// TwinCAT 3 PLC project Plc1_AmeClient
// ProgramVersion: 3.1.4024.0
// libraries:
//   Tc2_Standard, * (Beckhoff Automation GmbH)
//   Tc2_System, * (Beckhoff Automation GmbH)
//   Tc2_TcpIp, * (Beckhoff Automation GmbH)
//   Tc3_Module, * (Beckhoff Automation GmbH)
// project tree:
//   / PlcTask.TcTTO
//   POUs/AmeClient/ AmeClient.TcPOU (not stored), AmeClientParam.TcGVL (not stored)
//   POUs/AmeClient/DUTs/AssyMethods/ St_Assy_Base.TcDUT (not stored), St_Assy_Complete.TcDUT (not stored), St_Assy_GetDetails.TcDUT (not stored), St_Assy_SetParametricsAndNCNative.TcDUT (not stored), St_Assy_SetReferences.TcDUT (not stored), St_Assy_SignOff.TcDUT (not stored), St_Assy_Start.TcDUT (not stored)
//   POUs/AmeClient/DUTs/ E_AssyComplete.TcDUT (not stored)
//   POUs/ MAIN.TcPOU
//   POUs/OOP/ I_Command.TcIO (not stored), I_Device.TcIO (not stored), Stereo.TcPOU, TurnOffCommand.TcPOU (not stored), TurnOnCommand.TcPOU (not stored)
// real-time tasks:
//   TASK PlcTask: cycle T#10ms, priority 20, ADS port 350
// motion (NC):
//   TASK NC-Task 1 SAF: cycle T#2ms, priority 4, ADS port 501
//   TASK NC-Task 1 SVB: cycle T#10ms, priority 8, ADS port 511
//   AXIS Axis 1 (id 1)
//     OtherSettings: AllowMotionCmdToSlave=true
//     encoder EncType=19
//       EncPara: MaxCount=#xffffffff
//     drive DrvType=16
//       DrvPara: MaxCount=#xffffffff
//         Analog: TorqueSetpointScale=10, ScaleFactorActTorque=0.1
//         TimeComp: TaskDelayCycles=1
//     controller CtrType=1
//       CtrPara: PriorControlFactor=1
//         Observer: BandWidth=20
// I/O:
//   DEVICE Device 1 (EtherCAT) (disabled), AmsNetId 192.168.48.2.2.1
//     Term 1 (EK1100) [EK1100 EtherCAT Coupler (2A E-Bus)]
//       Term 2 (EL6631) [EL6631 PROFINET IO Controller]
//     ServoControllerX (CMMT-AS-MP-S1) [CMMT-AS-MP-S1]
//   DEVICE Device 2 (EL6631) (disabled), AmsNetId 192.168.48.2.3.1
//     tcpniodevice [Beckhoff Automation TwinCAT PLC PROFINET I/O Device with I/Os, V2.43, PROFIenergy supported; 1 port TwinCAT PN Device]
//       modules: Term 1 (DAP Module)
//     tcpniodevice-4 [Beckhoff Automation TwinCAT PLC PROFINET I/O Device with I/Os, V2.32, 1 port diagnostic supported TwinCAT PN Device]
//       modules: Term 2 (DAP Module), Term 3 (8 Word Output), Term 4 (2 Word Output), Term 5 (1 Word Output), Term 6 (1 Word Output), Term 7 (8 Word Input), Term 8 (2 Word Input), Term 9 (8 Word Input), Term 10 (64 Word Input)
// variable links:
//   (this object) <-> Device 1 (EtherCAT)/ServoControllerX (CMMT-AS-MP-S1)
//     Drive/Inputs/In/nDataIn3[0] <-> Inputs/Torque actual value
//     Drive/Inputs/In/nDcOutputTime <-> InfoData/DcOutputShift
//     Drive/Inputs/In/nState1 <-> Inputs/Statusword
//     Drive/Inputs/In/nState2 <-> Inputs/Statusword @bit 8
//     Drive/Inputs/In/nState4 @bit 1 <-> WcState/InputToggle
//     Drive/Inputs/In/nState4 <-> WcState/WcState
//     Drive/Inputs/In/nState5 <-> Inputs/Modes of operation display
//     Drive/Outputs/Out/nCtrl1 <-> Outputs/Controlword
//     Drive/Outputs/Out/nCtrl2 <-> Outputs/Controlword @bit 8
//     Drive/Outputs/Out/nCtrl5 <-> Outputs/Modes of operation
//     Drive/Outputs/Out/nDataOut1 <-> Outputs/Target position
//     Drive/Outputs/Out/nDataOut2 <-> Outputs/Target velocity
//     Drive/Outputs/Out/nDataOut3[0] <-> Outputs/Torque offset
//     Drive/Outputs/Out/nDataOut4[0] <-> Outputs/Target torque
//     Enc/Inputs/In/nDataIn1 <-> Inputs/Position actual value
//     Enc/Inputs/In/nDataIn7 <-> Inputs/Velocity actual value
//     Enc/Inputs/In/nDcInputTime <-> InfoData/DcInputShift
//     Enc/Inputs/In/nState4 @bit 1 <-> WcState/InputToggle
//     Enc/Inputs/In/nState4 <-> WcState/WcState

CONFIGURATION Plc1_AmeClient
    RESOURCE PLC ON TwinCAT3
        TASK PlcTask(INTERVAL := T#10ms, PRIORITY := 20);
        PROGRAM MAIN WITH PlcTask : MAIN;
    END_RESOURCE
END_CONFIGURATION

// ---- POUs/MAIN.TcPOU
PROGRAM MAIN

VAR	

	AmeClient 							:AmeClient(iType := 1, sSrvNetId := '', sRemoteHost := '192.168.48.2', udiRemotePort := 2001, tTimeout := T#5S);
	_bAssy_GetDetails 					:BOOL;
	_st_Assy_GetDetails					: St_Assy_GetDetails := (sSfc := 'TEST0100000000001010184E0010', iOpIndex := 0); 
	_bAssy_Start						:BOOL;
	_st_Assy_Start						:St_Assy_Start := (sSfc := 'TEST0100000000001010184E0010', iOpIndex := 0);
	_bAssy_SetReferences				:BOOL;
	_st_Assy_SetReferences				:St_Assy_SetReferences := (sSfc := 'TEST0100000000001010184E0010', sCustomField :='PLASMA_COUNTER|0',  iOpIndex := 0);
	_bAssy_SetParametricsAndNCNative	:BOOL;
	_st_Assy_SetParametricsAndNCNative	:St_Assy_SetParametricsAndNCNative := (	sSfc 			:= 'TEST0100000000001010184E0010',
																				sProgramId 		:= 'PROGRAMID_TEST1',
																				sProgramRevision:= 'PROGRAMREVISION_TEST1',
																				sTestStep		:= 'TESTESTEP1', 
																				sDescription	:= 'DESCRIPTION1', 
																				sValue			:= 'TESTVALUE1', 
																				sUnit			:= 'UNIT1', 
																				sLowerLimit		:= 'LOWERLIMIT1', 
																				sUpperLimit		:= 'UPPERLIMIT1', 
																				sState			:= '0', 
																				sAdapter		:= '2',
																				iOpIndex 		:= 0);
	_bAssy_Complete						:BOOL;
	_st_Assy_Complete					:St_Assy_Complete := (sSfc := 'TEST0100000000001010184E0010', eState := E_AssyComplete.PASS, iOpIndex := 0);
	_bAssy_SignOff						:BOOL;
	_st_Assy_SignOff					:St_Assy_SignOff := (sSfc := 'TEST0100000000001010184E0010', iOpIndex := 0);
	_sSendMsg							:STRING(AmeClientParam.udiMSG_SIZE);
	_sRcvMsg							:STRING(AmeClientParam.udiMSG_SIZE);
	
END_VAR

VAR
	bMsg	:Bool;
END_VAR

// Assy GetDetails******************************************************

IF(_bAssy_GetDetails = TRUE AND_THEN AmeClient.Assy_GetDetails_1026(_st_Assy_GetDetails) = TRUE) THEN
	_bAssy_GetDetails := FALSE;
	_sSendMsg 		:= AmeClient.sSendMsg;
	_sRcvMsg 		:= AmeClient.sRcvMsg;
END_IF
//**********************************************************************

// Assy Start***********************************************************
IF(_bAssy_Start = TRUE AND_THEN AmeClient.Assy_Start(_st_Assy_Start) = TRUE) THEN
	_bAssy_Start := FALSE;
	_sSendMsg 	:= AmeClient.sSendMsg;
	_sRcvMsg 	:= AmeClient.sRcvMsg;
END_IF
//**********************************************************************

// Assy setReferences***************************************************
IF(_bAssy_SetReferences = TRUE AND_THEN AmeClient.Assy_SetReferences_3026(_st_Assy_SetReferences) = TRUE ) THEN
	_bAssy_SetReferences := FALSE;
	_sSendMsg 	:= AmeClient.sSendMsg;
	_sRcvMsg 	:= AmeClient.sRcvMsg;
END_IF
//**********************************************************************

// Assy SetParametricsAndNCNative***************************************
IF(_bAssy_SetParametricsAndNCNative = TRUE AND_THEN AmeClient.Assy_SetParametricsAndNCNative_3503(_st_Assy_SetParametricsAndNCNative) = TRUE) THEN
	_bAssy_SetParametricsAndNCNative := FALSE;
	_sSendMsg 	:= AmeClient.sSendMsg;
	_sRcvMsg 	:= AmeClient.sRcvMsg;
END_IF
//**********************************************************************

// Assy compleate*******************************************************
IF(_bAssy_Complete = TRUE AND_THEN AmeClient.Assy_Complete_3011(_st_Assy_Complete) = TRUE) THEN
	_bAssy_Complete := FALSE;
	_sSendMsg := AmeClient.sSendMsg;
	_sRcvMsg := AmeClient.sRcvMsg;
END_IF
//**********************************************************************

// Assy signOff*********************************************************
IF(_bAssy_SignOff	 = TRUE AND_THEN AmeClient.Assy_SignOff(_st_Assy_SignOff) = TRUE) THEN
	_bAssy_SignOff	 := FALSE;
	_sSendMsg := AmeClient.sSendMsg;
	_sRcvMsg := AmeClient.sRcvMsg;
END_IF
//**********************************************************************

IF bMsg THEN
	ADSLOGSTR(msgCtrlMask := ADSLOG_MSGTYPE_LOG OR ADSLOG_MSGTYPE_LOG,
				msgFmtStr := 'Hello %s',
				strArg	:= 'world');
	bMsg := FALSE;
END_IF

END_PROGRAM

// ---- POUs/OOP/Stereo.TcPOU
FUNCTION_BLOCK Stereo IMPLEMENTS I_Device
VAR_INPUT
END_VAR
VAR_OUTPUT
END_VAR
VAR
END_VAR

METHOD adjustVolume
ADSLOGSTR(msgCtrlMask := ADSLOG_MSGTYPE_LOG OR ADSLOG_MSGTYPE_LOG,
		msgFmtStr := 'Volume adjusted',
		strArg	:= '');
END_METHOD

{warning 'add method implementation '}
METHOD turnOff
ADSLOGSTR(msgCtrlMask := ADSLOG_MSGTYPE_LOG OR ADSLOG_MSGTYPE_LOG,
		msgFmtStr := 'Stereo is now off',
		strArg	:= '');
END_METHOD

{warning 'add method implementation '}
METHOD turnOn
ADSLOGSTR(msgCtrlMask := ADSLOG_MSGTYPE_LOG OR ADSLOG_MSGTYPE_LOG,
		msgFmtStr := 'Stereo is now on',
		strArg	:= '');
END_METHOD

END_FUNCTION_BLOCK
